FUNCTION_BLOCK OPCUAC_18 (* 8-Channel OPC UA Client Interface Block *)
  (* Version 1.0, AN, SWDC RTSoft *)
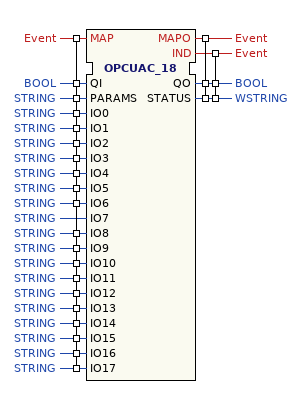
  EVENT_INPUT
    MAP WITH QI, PARAMS, IO0, IO1, IO2, IO3, IO4, IO5, IO6, IO8, IO9, IO10, IO11, IO12, IO13, IO14, IO15, IO16, IO17; (* Initialization Request *)
  END_EVENT
  EVENT_OUTPUT
    MAPO WITH QO, STATUS; (* Initialization Confirm *)
    IND WITH QO, STATUS; (* Execution Confirm *)
  END_EVENT
  VAR_INPUT
    QI : BOOL; (* Event Input Qualifier *)
    PARAMS : STRING; (* Initialization Parameters *)
    IO0 : STRING; (* Input Output 0 *)
    IO1 : STRING; (* Input Output 1 *)
    IO2 : STRING; (* Input Output 2 *)
    IO3 : STRING; (* Input Output 3 *)
    IO4 : STRING; (* Input Output 4 *)
    IO5 : STRING; (* Input Output 5 *)
    IO6 : STRING; (* Input Output 6 *)
    IO7 : STRING; (* Input Output 7 *)
    IO8 : STRING; (* Input Output 8 *)
    IO9 : STRING; (* Input Output 9 *)
    IO10 : STRING; (* Input Output 10 *)
    IO11 : STRING; (* Input Output 11 *)
    IO12 : STRING; (* Input Output 12 *)
    IO13 : STRING; (* Input Output 13 *)
    IO14 : STRING; (* Input Output 14 *)
    IO15 : STRING; (* Input Output 15 *)
    IO16 : STRING; (* Input Output 15 *)
    IO17 : STRING; (* Input Output 15 *)
  END_VAR
  VAR_OUTPUT
    QO : BOOL; (* Event Output Qualifier *)
    STATUS : WSTRING; (* Service Status *)
  END_VAR
END_FUNCTION_BLOCK
